INTERFACE I_HasErrorSourcing

PROPERTY ErrorSource : REFERENCE TO ST_ErrorSource
GET
END_GET
END_PROPERTY

END_INTERFACE

(* stored: Version 1.1.0.1, ProductVersion 3.1.4024.13
   Itf I_HasErrorSourcing: Id {eb5b0aa6-ca0e-0f30-0ce6-25eb6ff7d06b}
   Property ErrorSource: Id {c46375b7-659d-0834-28b0-bc5da84e87db}
   Get Get: Id {954df89a-cd7e-0384-3ae0-7a4699eb4eb0} *)
